VAR_GLOBAL CONSTANT
	cusiMinAddedChilds: USINT := 1;
	/// Buffer prepared for 80 sections, means, with section length e.g. 0.49 m a TLK with max. length of 39 m 
	cusiSectionBuffer_SIZE: USINT := 80;
END_VAR

(* stored: Version 1.1.0.1, ProductVersion 3.1.0.23
   GVL Const_MTR: Id {db967737-eb5b-4041-af96-2e99aca2b453} *)
